// TIA Portal project "Sorting_weight_Udemy_V19" (V19)

(* hardware
DEVICE "S7-1200 station_1"  S7-1200 Station
   slot 0: "Rack_0"  Rack  V1.0
   slot 1: "PLC_1"  CPU 1212C AC/DC/Rly  6ES7 212-1BE40-0XB0  V4.1
*)

// ===== PLC "PLC_1"  CPU 1212C AC/DC/Rly =====

VAR_GLOBAL   // PLC tag table "Default tag table"
   "Tag_1" AT %I50.0 : Bool;
   "Entry Conveyor" AT %Q0.0 : Bool;
   "Tag_3" AT %I0.0 : Bool;
   "Falling Edge" AT %M0.0 : Bool;
   "Tag_5" AT %ID30 : Real;
   "Entry sensor" AT %I0.1 : Bool;
   "Tag_7" AT %ID100 : Real;
   "Rising Edge1" AT %M0.1 : Bool;
   "Start" AT %I1.0 : Bool;
   "Roller forward" AT %Q0.1 : Bool;
   "Stop" AT %I1.1 : Bool;
   "Tag_2" AT %Q0.2 : Bool;
   "Tag_4" AT %Q0.3 : Bool;
   "Front Conveyor" AT %Q0.4 : Bool;
   "Left Conveyor" AT %Q0.5 : Bool;
   "Right COnveyor" AT %Q0.6 : Bool;
   "Load Scale" AT %Q0.7 : Bool;
   "Tag_13" AT %QD100 : DInt;
   "Exit left" AT %I0.2 : Bool;
   "Rising edge 2" AT %M0.2 : Bool;
   "Left count" AT %QD104 : DWord;
   "Exit right" AT %I0.3 : Bool;
   "Rising edge 3" AT %M0.3 : Bool;
   "Right Count" AT %QD108 : DWord;
   "Exit front" AT %I0.4 : Bool;
   "Rising Edge 4" AT %M0.4 : Bool;
   "Forward Count" AT %QD112 : DWord;
   "Reset Counts" AT %I1.2 : Bool;
   "Tag_17" AT %MB0 : Byte;
   "Tag_18" AT %MB5 : Byte;
   "Tag_19" AT %M50.0 : Bool;
   "Tag_20" AT %M50.1 : Bool;
   "Tag_6" AT %MB30 : Byte;
   "Tag_8" AT %I0.5 : Bool;
   "Tag_9" AT %M0.5 : Bool;
   "Tag_10" AT %MD30 : DWord;
   "Tag_11" AT %MW30 : Int;
   "Tag_12" AT %QD116 : DInt;
END_VAR

DATA_BLOCK "Weight"   // DB1
{ S7_Optimized_Access := 'TRUE' }
VERSION : 0.1
   VAR
      Weight : Array[0..2] of Real;
   END_VAR
BEGIN
END_DATA_BLOCK

// folder: System blocks/Program resources

DATA_BLOCK "IEC_Counter_0_DB"   // DB3
{ S7_Optimized_Access := 'TRUE' }
AUTHOR : Simatic
FAMILY : IEC
NAME : CNTR
VERSION : 1.0
// stored: InstanceOfName IEC_COUNTER
"IEC_COUNTER"
BEGIN
END_DATA_BLOCK

// folder: (top level)

FUNCTION "Block_1" : Void   // FC1, SCL
{ S7_Optimized_Access := 'TRUE' }
VERSION : 0.1
   VAR_INPUT
      recipe : Int;
      count : Int;   // present counts of counter
      weight : Real;   // sensor
      at_scale : Bool;   // on the sensor
   END_VAR
   VAR_OUTPUT
      "left roller" : Bool;
      "right roller" : Bool;
      weight_display : DInt;
      temp : Array[0..2] of Real;
   END_VAR
   VAR_TEMP
      Sorting : Array[0..5] of Bool;
   END_VAR
BEGIN
   //Recipe Logic
   IF #recipe = 0 THEN
       #Sorting[0] := 0;
       #Sorting[1] := 0;
       #Sorting[2] := 0;
       #Sorting[3] := 1;
       #Sorting[4] := 1;
       #Sorting[5] := 0;
   END_IF;

   IF #recipe = 1 THEN
       #Sorting[0] := 0;
       #Sorting[1] := 1;
       #Sorting[2] := 1;
       #Sorting[3] := 0;
       #Sorting[4] := 0;
       #Sorting[5] := 0;
   END_IF;

   IF #recipe = 2 THEN
       #Sorting[0] := 1;
       #Sorting[1] := 0;
       #Sorting[2] := 0;
       #Sorting[3] := 0;
       #Sorting[4] := 0;
       #Sorting[5] := 1;
   END_IF;

   IF #recipe > 2 OR #recipe < 0 THEN
       #recipe := 0;
   END_IF;

   //Storing Box information
   IF #at_scale = 1 THEN
       #temp[#count] := #weight;
   END_IF;

   //Large Box
   IF #temp[#count] > 7.0 AND #temp[#count] < 8.0 THEN
       #"left roller" := #Sorting[0];
       #"right roller" := #Sorting[1];
   END_IF;

   //Medium Box
   IF #temp[#count] > 4.5 AND #temp[#count] < 5.5 THEN
       #"left roller" := #Sorting[2];
       #"right roller" := #Sorting[3];
   END_IF;

   //Small Box
   IF #temp[#count] > 3.5 AND #temp[#count] < 4.5 THEN
       #"left roller" := #Sorting[4];
       #"right roller" := #Sorting[5];
   END_IF;
   //For displaying Weight on Panel
   #weight_display := REAL_TO_DINT(#weight * 10.0) ;
END_FUNCTION

ORGANIZATION_BLOCK "Main"   // OB1, LAD, ProgramCycle
TITLE = "Main Program Sweep (Cycle)"
{ S7_Optimized_Access := 'TRUE' }
VERSION : 0.1
   VAR_INPUT
      Initial_Call : Bool;   // Initial call of this OB
      Remanence : Bool;   // =True, if remanent data are available
   END_VAR
   VAR_TEMP   // added for the SCL form of the ladder/FBD networks
      _w1 : Bool;
   END_VAR
BEGIN

REGION Network 1: Start/Stop main Conveyor
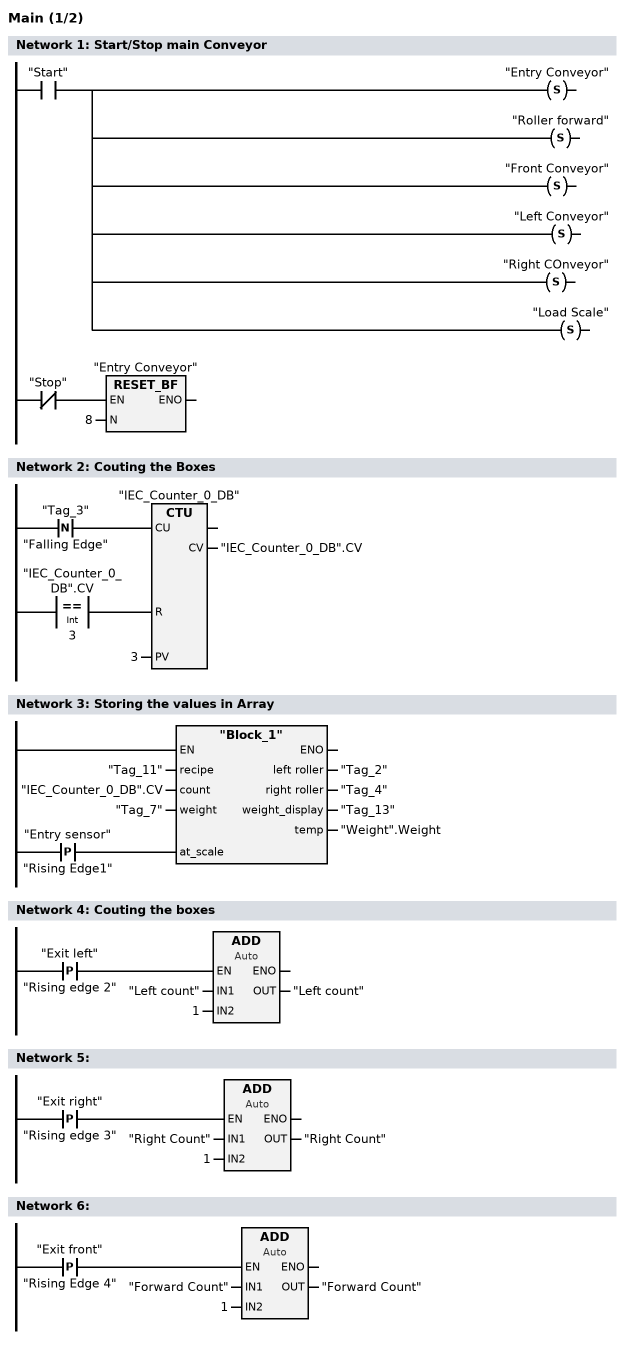
   // no SCL statement known for RBitfield: written as a call
   IF "Start" THEN
       "Entry Conveyor" := TRUE;
       "Roller forward" := TRUE;
       "Front Conveyor" := TRUE;
       "Left Conveyor" := TRUE;
       "Right COnveyor" := TRUE;
       "Load Scale" := TRUE;
   END_IF;
   IF NOT "Stop" THEN RESET_BF(operand := "Entry Conveyor", n := 8); END_IF;
END_REGION

REGION Network 2: Couting the Boxes
   #_w1 := NOT "Tag_3" AND "Falling Edge";   // falling edge of "Tag_3"
   "Falling Edge" := "Tag_3";
   "IEC_Counter_0_DB".CTU(CU := #_w1, R := "IEC_Counter_0_DB".CV = 3, PV := 3, CV => "IEC_Counter_0_DB".CV);
END_REGION

REGION Network 3: Storing the values in Array
   RUNG wire#powerrail
      "Block_1"(at_scale := wire#w1, recipe := "Tag_11", count := "IEC_Counter_0_DB".CV, weight := "Tag_7", "left roller" => "Tag_2", "right roller" => "Tag_4", weight_display => "Tag_13", temp => "Weight".Weight)
   END_RUNG
   RUNG wire#powerrail
      P_Contact(operand := "Entry sensor", bit := "Rising Edge1")
   END_RUNG wire#w1
   // the same network as SCL:
   #_w1 := "Entry sensor" AND NOT "Rising Edge1";   // rising edge of "Entry sensor"
   "Rising Edge1" := "Entry sensor";
   "Block_1"(recipe := "Tag_11",
             count := "IEC_Counter_0_DB".CV,
             weight := "Tag_7",
             at_scale := #_w1,
             "left roller" => "Tag_2",
             "right roller" => "Tag_4",
             weight_display => "Tag_13",
             temp => "Weight".Weight);
END_REGION

REGION Network 4: Couting the boxes
   RUNG wire#powerrail
      P_Contact(operand := "Exit left", bit := "Rising edge 2")
      { S7_GenerateENO := "TRUE" } Add(in1 := "Left count", in2 := 1, out => "Left count")
   END_RUNG
   // the same network as SCL:
   #_w1 := "Exit left" AND NOT "Rising edge 2";   // rising edge of "Exit left"
   "Rising edge 2" := "Exit left";
   IF #_w1 THEN "Left count" := "Left count" + 1; END_IF;
END_REGION

REGION Network 5
   RUNG wire#powerrail
      P_Contact(operand := "Exit right", bit := "Rising edge 3")
      { S7_GenerateENO := "TRUE" } Add(in1 := "Right Count", in2 := 1, out => "Right Count")
   END_RUNG
   // the same network as SCL:
   #_w1 := "Exit right" AND NOT "Rising edge 3";   // rising edge of "Exit right"
   "Rising edge 3" := "Exit right";
   IF #_w1 THEN "Right Count" := "Right Count" + 1; END_IF;
END_REGION

REGION Network 6
   RUNG wire#powerrail
      P_Contact(operand := "Exit front", bit := "Rising Edge 4")
      { S7_GenerateENO := "TRUE" } Add(in1 := "Forward Count", in2 := 1, out => "Forward Count")
   END_RUNG
   // the same network as SCL:
   #_w1 := "Exit front" AND NOT "Rising Edge 4";   // rising edge of "Exit front"
   "Rising Edge 4" := "Exit front";
   IF #_w1 THEN "Forward Count" := "Forward Count" + 1; END_IF;
END_REGION

REGION Network 7
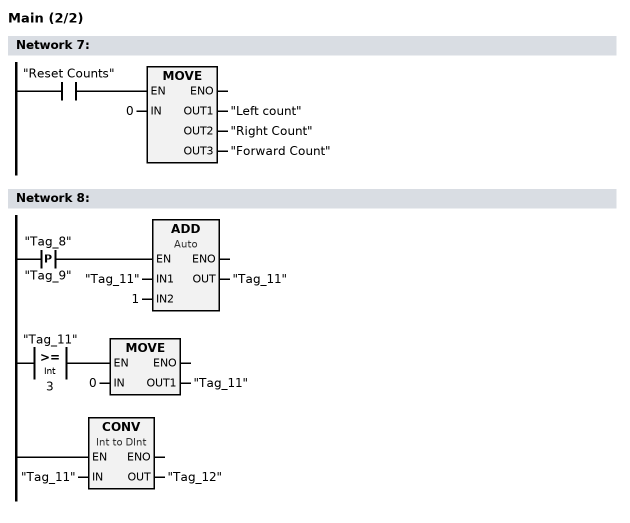
   RUNG wire#powerrail
      Contact( "Reset Counts" )
      { S7_GenerateENO := "TRUE" } Move(in := 0, out1 => "Left count", out2 => "Right Count", out3 => "Forward Count")
   END_RUNG
   // the same network as SCL:
   IF "Reset Counts" THEN
       "Left count" := 0;
       "Right Count" := 0;
       "Forward Count" := 0;
   END_IF;
END_REGION

REGION Network 8
   RUNG wire#powerrail
      P_Contact(operand := "Tag_8", bit := "Tag_9")
      { S7_GenerateENO := "TRUE" } Add(in1 := "Tag_11", in2 := 1, out => "Tag_11")
   END_RUNG
   RUNG wire#powerrail
      { S7_Templates := "SrcType := Int" } GE_Contact(in1 := "Tag_11", in2 := 3)
      { S7_GenerateENO := "TRUE" } Move(in := 0, out1 => "Tag_11")
   END_RUNG
   RUNG wire#powerrail
      { S7_Templates := "[SrcType := Int, DestType := DInt]"; S7_GenerateENO := "TRUE" } Convert(in := "Tag_11", out => "Tag_12")
   END_RUNG
   // the same network as SCL:
   #_w1 := "Tag_8" AND NOT "Tag_9";   // rising edge of "Tag_8"
   "Tag_9" := "Tag_8";
   IF #_w1 THEN "Tag_11" := "Tag_11" + 1; END_IF;
   IF "Tag_11" >= 3 THEN "Tag_11" := 0; END_IF;
   "Tag_12" := INT_TO_DINT("Tag_11");
END_REGION
END_ORGANIZATION_BLOCK